{attribute 'qualified_only'}
VAR_GLOBAL
  runner: EventRunner;
END_VAR

(* stored: Version 1.1.0.1, ProductVersion 3.1.4024.9
   GVL GVL: Id {e8cbc2c7-be2b-47ec-9cc7-f499f2cc99d1} *)
